ADAPTER ILevelFeedFlow (* Adapter Interface *)
  (* Standard: 61499-1 *)
  (* Version 0.0, 9/23/2026, Schneider Electric *)
  PACKAGE SE.Nereda;
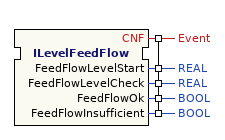
  EVENT_OUTPUT
    CNF WITH FeedFlowLevelStart, FeedFlowLevelCheck, FeedFlowOk, FeedFlowInsufficient; (* Confirmation from Plug *)
  END_EVENT
  VAR_OUTPUT
    FeedFlowLevelStart : REAL;
    FeedFlowLevelCheck : REAL;
    FeedFlowOk : BOOL;
    FeedFlowInsufficient : BOOL;
  END_VAR
  SERVICE SOCKET/PLUG
    SEQUENCE request_confirm
      SOCKET.REQ(REQD) -> PLUG.REQ(REQD);
      PLUG.CNF(CNFD) -> SOCKET.CNF(CNFD);
    END_SEQUENCE
    SEQUENCE indication_response
      PLUG.IND(INDD) -> SOCKET.IND(INDD);
      SOCKET.RSP(RSPD) -> PLUG.RSP(RSPD);
    END_SEQUENCE
  END_SERVICE
END_ADAPTER
